// TIA Portal V17 export
// export: Created 2023-02-14T02:49:13.871729Z, ExportSetting WithDefaults, DisplayName Totally Integrated Automation Portal, DisplayVersion V17, DisplayName TIA Portal Openness, DisplayVersion V17, DisplayName TIA Portal Teamcenter Gateway, DisplayVersion V17, DisplayName TIA Portal Version Control Interface, DisplayVersion V17, DisplayName SINAMICS Startdrive Advanced, DisplayVersion V17, DisplayName SINAMICS Startdrive G130, G150, S120, S150, SINAMICS MV, S210, DisplayVersion V17, DisplayName SINAMICS Startdrive G110M, G120, G120C, G120D, G120P, G115D, DisplayVersion V17, DisplayName STEP 7 Professional, DisplayVersion V17, DisplayName STEP 7 Safety, DisplayVersion V17, DisplayName WinCC Professional, DisplayVersion V17
DATA_BLOCK "THE-1 to Stock Tank"   // DB452
{ S7_Optimized_Access := 'FALSE' }
VERSION : 0.1
// stored: AutoNumber false, DBAccessibleFromOPCUA true, DBAccessibleFromWebserver true, IsOnlyStoredInLoadMemory false, IsWriteProtectedInAS false
   VAR
      CIP_Request : Bool;
      free_bool_2 : Bool;
      free_bool_3 : Bool;
      free_bool_4 : Bool;
      free_bool_5 : Bool;
      free_bool_6 : Bool;
      free_bool_7 : Bool;
      free_bool_8 : Bool;
      free_bool_9 : Bool;
      free_bool_10 : Bool;
      free_bool_11 : Bool;
      free_bool_12 : Bool;
      free_bool_13 : Bool;
      free_bool_14 : Bool;
      free_bool_15 : Bool;
      free_bool_16 : Bool;
      free_real_1 : Real;
      free_real_2 : Real;
      free_real_3 : Real;
      free_real_4 : Real;
      free_real_5 : Real;
      free_real_6 : Real;
      free_real_7 : Real;
      free_real_8 : Real;
      free_byte_1 : Byte;
      free_byte_2 : Byte;
      free_byte_3 : Byte;
      free_byte_4 : Byte;
      free_byte_5 : Byte;
      free_byte_6 : Byte;
      free_byte_7 : Byte;
      free_byte_8 : Byte;
   END_VAR
BEGIN
END_DATA_BLOCK
